// TIA Portal V19 export
FUNCTION_BLOCK "Positioning_EPOS_Machine_FB"   // FB55, LAD
TITLE = CLOSE LOOP POSITIONING AXIS WITH DRIVE S120 TEL.111 EPOS
// stored: Access Published, MemoryReserve 100, SetENOAutomatically false
   VAR_INPUT
      AreaInterface : "AreaInterface";
      ZSI : "udt_ZoneSafetyInterface";
      DSI : "udt_DeviceSafetyInterface";
      Drive : "TAx_DriveInterface";
      DataIn : "Positioning_EPOS_Machine_DataIn";
      CIn : "Positioning_EPOS_Machine_CIn";
      Config : "Positioning_EPOS_Machine_Config";
      HW_ID_TEL111 : HW_SUBMODULE;
   END_VAR
   VAR_OUTPUT
      MachineInterface { ExternalAccessible := 'False'; ExternalVisible := 'False'; ExternalWritable := 'False'} : "MachineInterface";
      DataOut : "Positioning_EPOS_Machine_DataOut";
      COut : "Positioning_EPOS_Machine_COut";
   END_VAR
   VAR_IN_OUT
      Par : "Positioning_EPOS_Machine_Par";
      Warning : "Positioning_EPOS_Machine_Wng";
      Alarm : "Positioning_EPOS_Machine_Alr";
   END_VAR
   VAR
      InitDone : Bool := FALSE;
      Status : Int;
      Diag : Struct
         S120 : "TO_Diagnostic";
      END_STRUCT;
      HMI : Struct
         Sts { S7_SetPoint := 'True'} : "UDT_HMI-Sts_PosEPOS-MchFB";
         B_Preset : Bool;
         PresetPosition : LReal;
         TargetPosition : LReal;
      END_STRUCT;
      Sts : Struct
         Standstill : Bool;
         AlarmPresence : Bool;
         WarningPresence : Bool;
         Gen_Cnd : Bool;
         Minus_Cnd : Bool;
         Plus_Cnd : Bool;
         Pos_Cnd : Bool;
         Preset_Cnd : Bool;
         InTargetPosition : Bool;
         Limits_SW_Active : Bool;
         Limits_EXT_Active : Bool;
         AxisModulo : LReal;
         ActualPosition : LReal;
         MissingToTarget : LReal;
         ActualVelocityRPM : LReal;
         ReductionRatio : LReal;
         ActualVelocity : LReal;
         S120 : Struct
            FaultActive : Bool;
            AlarmPresence : Bool;
            Standstill : Bool;
            IsRunningNegative : Bool;
            IsRunningPositive : Bool;
            MinusSWLim : Bool;
            PlusSWLim : Bool;
            MinusHWLim : Bool;
            PlusHWLim : Bool;
            TargetApply : Bool;
         END_STRUCT;
      END_STRUCT;
      Ctrl : Struct
         StopDueDoorOpeningRequest : Bool;
         StopAborting : Bool;
         SafeMotionEnable : Bool;
         StopInPhase : Bool;
         StopProgrammed : Bool;
         Preset : Bool;
         Minus_Man : Bool;
         Plus_Man : Bool;
         MoveToPos_Man : Bool;
         Minus_Aut : Bool;
         Plus_Aut : Bool;
         MoveToPos_Aut : Bool;
         MoveToPos : Bool;
         Minus_Vel : Bool;
         Plus_Vel : Bool;
         Fan : Bool;
         Pos : LReal;
         Vel : LReal;
         Acc : LReal;
         Dec : LReal;
         S120 : Struct
            Preset : Bool;
            Jog_Plus : Bool;
            Jog_Minus : Bool;
            Positioining : Bool;
            TargetPos : DInt;   // [LU] = Eng.Unit / 1000
         END_STRUCT;
      END_STRUCT;
      S120_SinaPos { S7_SetPoint := 'True'} : SinaPos;
      Fan_M : "Motor";
      WriteRefPos { S7_SetPoint := 'True'} : "RW_SINAMICS_Par";
      TON_DelayOFF { S7_SetPoint := 'True'} : TON_TIME;
      TON_ModeTimeOut { S7_SetPoint := 'True'} : TON_TIME;
      TON_NoPendingCmd : TON_TIME;
      TON_MinusCnd { S7_SetPoint := 'True'} : TON_TIME;
      TON_PlusCnd { S7_SetPoint := 'True'} : TON_TIME;
      TON_Fan_DelayOff : TON_TIME;
      TON_Brake_TimeOut : TON_TIME;
      TON_InTargetPosition { S7_SetPoint := 'True'} : TON_TIME;
      AUX : Struct
         PB_Minus : Bool;
         PB_Plus : Bool;
         PB_MoveToPos { ExternalAccessible := 'False'; ExternalVisible := 'False'; ExternalWritable := 'False'} : Bool;
         B_Preset { ExternalAccessible := 'False'; ExternalVisible := 'False'; ExternalWritable := 'False'} : Bool;
      END_STRUCT;
   END_VAR
   VAR_TEMP
      PE : Struct
         PB_Minus : Bool;
         PB_Plus : Bool;
         PB_MoveToPos : Bool;
         B_Preset : Bool;
      END_STRUCT;
      RETVAL : Int;
      Req : Bool;
      RemainingDistanceABS : LReal;
      LimitExceeds : Bool;
      UsePositionLimits : Bool;
      DriveSwitchOnInhibit : Bool;
   END_VAR
   VAR CONSTANT
      MODE_1_RELATIVE_POSITIONING : Int := 1;
      MODE_2_ABSOLUTE_POSITIONING : Int := 2;
      MODE_3_POS_AS_SETUP : Int := 3;
      MODE_4_HOMING_PROCEDURE : Int := 4;
      MODE_5_SET_HOME_POSITION : Int := 5;
      MODE_6_TRAVERSING_BLOCK : Int := 6;
      MODE_7_JOG : Int := 7;
      MODE_8_JOG_INCREMENTAL : Int := 8;
      STS_0_IDLE : Int := 0;
      STS_DIRECT_HOME : Int := 10;
      STS_MOVE_VEL : Int := 20;
      STS_POSITIONING_START : Int := 30;
      STS_STOP : Int := 90;
   END_VAR
   VAR_TEMP   // added for the SCL form of the ladder/FBD networks
      _w1 : Bool;
      _w2 : Bool;
      _w3 : Bool;
      _w4 : Bool;
   END_VAR
BEGIN

REGION Network 1 (SCL): Init

   IF NOT #InitDone THEN

       #InitDone := TRUE;

   END_IF;
END_REGION

REGION Network 2 (SCL): Reset
   IF #AreaInterface.RstAlarms THEN


       #Alarm.Ax_NotHomed := FALSE;
       #Alarm.HwLimitMinus := FALSE;
       #Alarm.HwLimitPlus := FALSE;


       #Warning.NotAutReady := FALSE;
       #Warning.Minus_CndMissing := FALSE;
       #Warning.Plus_CndMissing := FALSE;



   END_IF;
END_REGION

REGION Network 3: Reduction ratio calculation - Motor revolution -> position Eng Unit
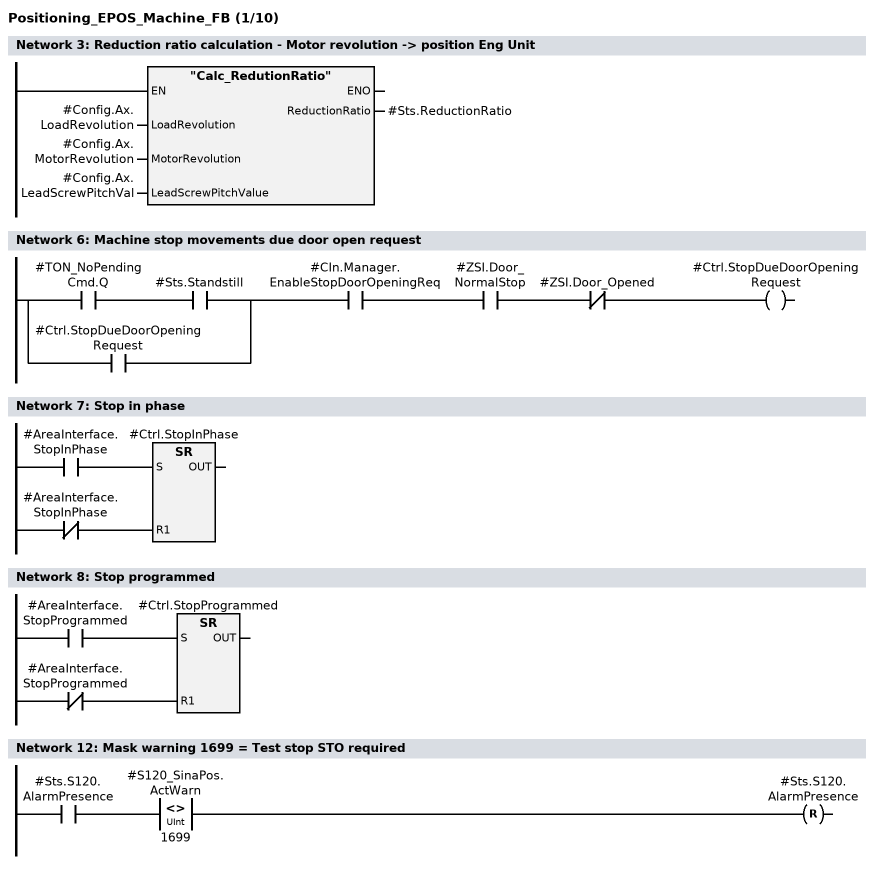
   RUNG wire#powerrail
      "Calc_RedutionRatio"(LoadRevolution := #Config.Ax.LoadRevolution, MotorRevolution := #Config.Ax.MotorRevolution, LeadScrewPitchValue := #Config.Ax.LeadScrewPitchVal, ReductionRatio => #Sts.ReductionRatio)
   END_RUNG
   // the same network as SCL:
   "Calc_RedutionRatio"(LoadRevolution := #Config.Ax.LoadRevolution,
                        MotorRevolution := #Config.Ax.MotorRevolution,
                        LeadScrewPitchValue := #Config.Ax.LeadScrewPitchVal,
                        ReductionRatio => #Sts.ReductionRatio);
END_REGION

REGION Network 4: >
END_REGION

REGION Network 5: <<< MACHINE STOP >>>
END_REGION

REGION Network 6: Machine stop movements due door open request
   RUNG wire#powerrail
      Contact( #TON_NoPendingCmd.Q )
      Contact( #Sts.Standstill )
      wire#w1
      Contact( #CIn.Manager.EnableStopDoorOpeningReq )
      Contact( #ZSI.Door_NormalStop )
      I_Contact( #ZSI.Door_Opened )
      Coil( #Ctrl.StopDueDoorOpeningRequest )
   END_RUNG
   RUNG wire#powerrail
      Contact( #Ctrl.StopDueDoorOpeningRequest )
   END_RUNG wire#w1
   // the same network as SCL:
   #Ctrl.StopDueDoorOpeningRequest := ((#TON_NoPendingCmd.Q AND #Sts.Standstill) OR #Ctrl.StopDueDoorOpeningRequest) AND #CIn.Manager.EnableStopDoorOpeningReq AND #ZSI.Door_NormalStop AND NOT #ZSI.Door_Opened;
END_REGION

REGION Network 7: Stop in phase
   RUNG wire#powerrail
      Contact( #AreaInterface.StopInPhase )
      S_SR(operand := #Ctrl.StopInPhase, r1 := wire#w1)
   END_RUNG
   RUNG wire#powerrail
      I_Contact( #AreaInterface.StopInPhase )
   END_RUNG wire#w1
   // the same network as SCL:
   IF #AreaInterface.StopInPhase THEN
       #Ctrl.StopInPhase := TRUE;   // SR flip-flop
   END_IF;
   IF NOT #AreaInterface.StopInPhase THEN #Ctrl.StopInPhase := FALSE; END_IF;
END_REGION

REGION Network 8: Stop programmed
   RUNG wire#powerrail
      Contact( #AreaInterface.StopProgrammed )
      S_SR(operand := #Ctrl.StopProgrammed, r1 := wire#w1)
   END_RUNG
   RUNG wire#powerrail
      I_Contact( #AreaInterface.StopProgrammed )
   END_RUNG wire#w1
   // the same network as SCL:
   IF #AreaInterface.StopProgrammed THEN
       #Ctrl.StopProgrammed := TRUE;   // SR flip-flop
   END_IF;
   IF NOT #AreaInterface.StopProgrammed THEN #Ctrl.StopProgrammed := FALSE; END_IF;
END_REGION

REGION Network 9: >
END_REGION

REGION Network 10 (SCL): Several status from FB
   // Axis modulo in Eng.Unit of position
   // 
   #Sts.AxisModulo := #Config.Ax.Modulo_S120_P2566 / 1000.0;


   // Position in Eng.Unit = Position in LU X 1000.
   //
   #Sts.ActualPosition := DINT_TO_LREAL(#S120_SinaPos.ActPosition) / 1000.0;

   // S120_SinaPos.ActVelocity = Current velocity (standardized 40000000h = 1073741824.0 dec = 100% = p2000)
   // Velocity in RPM
   // 
   #Sts.ActualVelocityRPM := DINT_TO_LREAL(#S120_SinaPos.ActVelocity) / 1073741824.0 * #Config.Ax.MaxRPM_S120_P2000;

   // Velocity in Eng.Unit / min
   #Sts.ActualVelocity := #Sts.ActualVelocityRPM * #Sts.ReductionRatio;


   #Sts.S120.IsRunningPositive := #S120_SinaPos.EPosZSW2.%X4;
   #Sts.S120.IsRunningNegative := #S120_SinaPos.EPosZSW2.%X5;

   #Sts.S120.MinusSWLim := #S120_SinaPos.EPosZSW2.%X6;
   #Sts.S120.PlusSWLim := #S120_SinaPos.EPosZSW2.%X7;

   #Sts.S120.MinusHWLim := #S120_SinaPos.EPosZSW1.%X8;
   #Sts.S120.PlusHWLim :=  #S120_SinaPos.EPosZSW1.%X9;


   #Sts.S120.FaultActive := #S120_SinaPos.ZSW1.%X3;
   #Sts.S120.AlarmPresence := #S120_SinaPos.ZSW1.%X7;
   #Sts.S120.Standstill := NOT #S120_SinaPos.EPosZSW1.%X4 AND NOT #S120_SinaPos.EPosZSW1.%X5 AND NOT #S120_SinaPos.EPosZSW2.%X4 AND NOT #S120_SinaPos.EPosZSW2.%X5;
END_REGION

REGION Network 11 (SCL): Drive Diagnostic
   #Diag.S120.DeviceType := 6;


   #Diag.S120.Drive_Message := 0;
   #Diag.S120.MessageType := 0;


   IF #Sts.S120.FaultActive THEN
       #Diag.S120.Drive_Message := #S120_SinaPos.ActFault;
       #Diag.S120.MessageType := 2;

   ELSIF #Sts.S120.AlarmPresence THEN
       #Diag.S120.Drive_Message := #S120_SinaPos.ActWarn;
       #Diag.S120.MessageType := 1;
   END_IF;
END_REGION

REGION Network 12: Mask warning 1699 = Test stop STO required
   RUNG wire#powerrail
      Contact( #Sts.S120.AlarmPresence )
      { S7_Templates := "SrcType := UInt" } NE_Contact(in1 := #S120_SinaPos.ActWarn, in2 := 1699)
      R_Coil( #Sts.S120.AlarmPresence )
   END_RUNG
   // the same network as SCL:
   IF #Sts.S120.AlarmPresence AND (#S120_SinaPos.ActWarn <> 1699) THEN
       #Sts.S120.AlarmPresence := FALSE;
   END_IF;
END_REGION

REGION Network 13: Drive / Axis Warnings
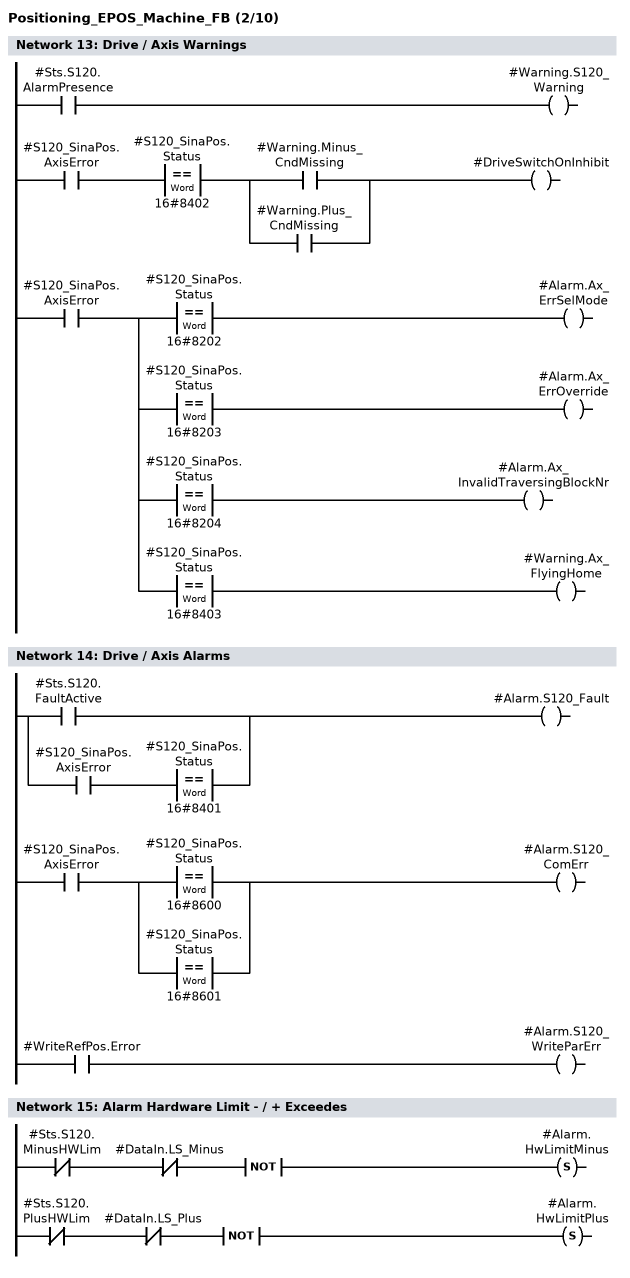
   RUNG wire#powerrail
      Contact( #Sts.S120.AlarmPresence )
      Coil( #Warning.S120_Warning )
   END_RUNG
   RUNG wire#powerrail
      Contact( #S120_SinaPos.AxisError )
      { S7_Templates := "SrcType := Word" } EQ_Contact(in1 := #S120_SinaPos.Status, in2 := 16#8402)
      wire#w1
      Contact( #Warning.Minus_CndMissing )
      wire#w2
      Coil( #DriveSwitchOnInhibit )
   END_RUNG
   RUNG wire#w1
      Contact( #Warning.Plus_CndMissing )
   END_RUNG wire#w2
   RUNG wire#powerrail
      Contact( #S120_SinaPos.AxisError )
      wire#w3
      { S7_Templates := "SrcType := Word" } EQ_Contact(in1 := #S120_SinaPos.Status, in2 := 16#8202)
      Coil( #Alarm.Ax_ErrSelMode )
   END_RUNG
   RUNG wire#w3
      { S7_Templates := "SrcType := Word" } EQ_Contact(in1 := #S120_SinaPos.Status, in2 := 16#8203)
      Coil( #Alarm.Ax_ErrOverride )
   END_RUNG
   RUNG wire#w3
      { S7_Templates := "SrcType := Word" } EQ_Contact(in1 := #S120_SinaPos.Status, in2 := 16#8204)
      Coil( #Alarm.Ax_InvalidTraversingBlockNr )
   END_RUNG
   RUNG wire#w3
      { S7_Templates := "SrcType := Word" } EQ_Contact(in1 := #S120_SinaPos.Status, in2 := 16#8403)
      Coil( #Warning.Ax_FlyingHome )
   END_RUNG
   // the same network as SCL:
   #Warning.S120_Warning := #Sts.S120.AlarmPresence;
   #DriveSwitchOnInhibit := #S120_SinaPos.AxisError AND (#S120_SinaPos.Status = 16#8402) AND (#Warning.Minus_CndMissing OR #Warning.Plus_CndMissing);
   #Alarm.Ax_ErrSelMode := #S120_SinaPos.AxisError AND (#S120_SinaPos.Status = 16#8202);
   #Alarm.Ax_ErrOverride := #S120_SinaPos.AxisError AND (#S120_SinaPos.Status = 16#8203);
   #Alarm.Ax_InvalidTraversingBlockNr := #S120_SinaPos.AxisError AND (#S120_SinaPos.Status = 16#8204);
   #Warning.Ax_FlyingHome := #S120_SinaPos.AxisError AND (#S120_SinaPos.Status = 16#8403);
END_REGION

REGION Network 14: Drive / Axis Alarms
   RUNG wire#powerrail
      Contact( #Sts.S120.FaultActive )
      wire#w1
      Coil( #Alarm.S120_Fault )
   END_RUNG
   RUNG wire#powerrail
      Contact( #S120_SinaPos.AxisError )
      { S7_Templates := "SrcType := Word" } EQ_Contact(in1 := #S120_SinaPos.Status, in2 := 16#8401)
   END_RUNG wire#w1
   RUNG wire#powerrail
      Contact( #S120_SinaPos.AxisError )
      wire#w2
      { S7_Templates := "SrcType := Word" } EQ_Contact(in1 := #S120_SinaPos.Status, in2 := 16#8600)
      wire#w3
      Coil( #Alarm.S120_ComErr )
   END_RUNG
   RUNG wire#w2
      { S7_Templates := "SrcType := Word" } EQ_Contact(in1 := #S120_SinaPos.Status, in2 := 16#8601)
   END_RUNG wire#w3
   RUNG wire#powerrail
      Contact( #WriteRefPos.Error )
      Coil( #Alarm.S120_WriteParErr )
   END_RUNG
   // the same network as SCL:
   #Alarm.S120_Fault := #Sts.S120.FaultActive OR (#S120_SinaPos.AxisError AND (#S120_SinaPos.Status = 16#8401));
   #Alarm.S120_ComErr := #S120_SinaPos.AxisError AND ((#S120_SinaPos.Status = 16#8600) OR (#S120_SinaPos.Status = 16#8601));
   #Alarm.S120_WriteParErr := #WriteRefPos.Error;
END_REGION

REGION Network 15: Alarm Hardware Limit - / + Exceedes
   RUNG wire#powerrail
      I_Contact( #Sts.S120.MinusHWLim )
      I_Contact( #DataIn.LS_Minus )
      Not()
      S_Coil( #Alarm.HwLimitMinus )
   END_RUNG
   RUNG wire#powerrail
      I_Contact( #Sts.S120.PlusHWLim )
      I_Contact( #DataIn.LS_Plus )
      Not()
      S_Coil( #Alarm.HwLimitPlus )
   END_RUNG
   // the same network as SCL:
   IF NOT (NOT #Sts.S120.MinusHWLim AND NOT #DataIn.LS_Minus) THEN #Alarm.HwLimitMinus := TRUE; END_IF;
   IF NOT (NOT #Sts.S120.PlusHWLim AND NOT #DataIn.LS_Plus) THEN #Alarm.HwLimitPlus := TRUE; END_IF;
END_REGION

REGION Network 16: Warning software limit - / + Exceedes
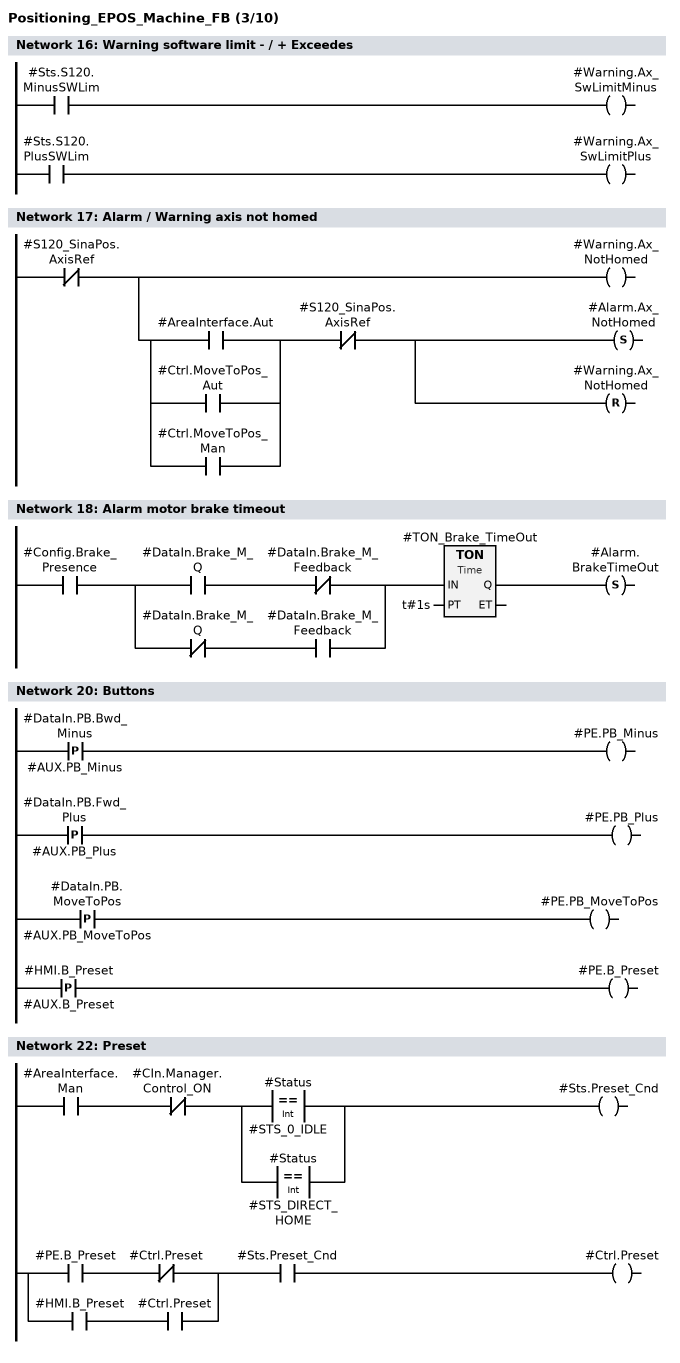
   RUNG wire#powerrail
      Contact( #Sts.S120.MinusSWLim )
      Coil( #Warning.Ax_SwLimitMinus )
   END_RUNG
   RUNG wire#powerrail
      Contact( #Sts.S120.PlusSWLim )
      Coil( #Warning.Ax_SwLimitPlus )
   END_RUNG
   // the same network as SCL:
   #Warning.Ax_SwLimitMinus := #Sts.S120.MinusSWLim;
   #Warning.Ax_SwLimitPlus := #Sts.S120.PlusSWLim;
END_REGION

REGION Network 17: Alarm / Warning axis not homed
   RUNG wire#powerrail
      I_Contact( #S120_SinaPos.AxisRef )
      wire#w1
      Coil( #Warning.Ax_NotHomed )
   END_RUNG
   RUNG wire#w1
      Contact( #AreaInterface.Aut )
      wire#w2
      I_Contact( #S120_SinaPos.AxisRef )
      wire#w3
      S_Coil( #Alarm.Ax_NotHomed )
   END_RUNG
   RUNG wire#w1
      Contact( #Ctrl.MoveToPos_Aut )
   END_RUNG wire#w2
   RUNG wire#w1
      Contact( #Ctrl.MoveToPos_Man )
   END_RUNG wire#w2
   RUNG wire#w3
      R_Coil( #Warning.Ax_NotHomed )
   END_RUNG
   // the same network as SCL:
   #Warning.Ax_NotHomed := NOT #S120_SinaPos.AxisRef;
   IF NOT #S120_SinaPos.AxisRef AND (#AreaInterface.Aut OR #Ctrl.MoveToPos_Aut OR #Ctrl.MoveToPos_Man) AND NOT #S120_SinaPos.AxisRef THEN
       #Alarm.Ax_NotHomed := TRUE;
       #Warning.Ax_NotHomed := FALSE;
   END_IF;
END_REGION

REGION Network 18: Alarm motor brake timeout
   RUNG wire#powerrail
      Contact( #Config.Brake_Presence )
      wire#w1
      Contact( #DataIn.Brake_M_Q )
      I_Contact( #DataIn.Brake_M_Feedback )
      wire#w2
      { S7_Templates := "time_type := Time" } #TON_Brake_TimeOut.TON(pt := t#1s, et =>)
      S_Coil( #Alarm.BrakeTimeOut )
   END_RUNG
   RUNG wire#w1
      I_Contact( #DataIn.Brake_M_Q )
      Contact( #DataIn.Brake_M_Feedback )
   END_RUNG wire#w2
   // the same network as SCL:
   #TON_Brake_TimeOut(IN := #Config.Brake_Presence AND ((#DataIn.Brake_M_Q AND NOT #DataIn.Brake_M_Feedback) OR (NOT #DataIn.Brake_M_Q AND #DataIn.Brake_M_Feedback)),   // TON
                      PT := t#1s);
   IF #TON_Brake_TimeOut.Q THEN #Alarm.BrakeTimeOut := TRUE; END_IF;
END_REGION

REGION Network 19: >
END_REGION

REGION Network 20: Buttons
   RUNG wire#powerrail
      P_Contact(operand := #DataIn.PB.Bwd_Minus, bit := #AUX.PB_Minus)
      Coil( #PE.PB_Minus )
   END_RUNG
   RUNG wire#powerrail
      P_Contact(operand := #DataIn.PB.Fwd_Plus, bit := #AUX.PB_Plus)
      Coil( #PE.PB_Plus )
   END_RUNG
   RUNG wire#powerrail
      P_Contact(operand := #DataIn.PB.MoveToPos, bit := #AUX.PB_MoveToPos)
      Coil( #PE.PB_MoveToPos )
   END_RUNG
   RUNG wire#powerrail
      P_Contact(operand := #HMI.B_Preset, bit := #AUX.B_Preset)
      Coil( #PE.B_Preset )
   END_RUNG
   // the same network as SCL:
   #_w1 := #DataIn.PB.Bwd_Minus AND NOT #AUX.PB_Minus;   // rising edge of #DataIn.PB.Bwd_Minus
   #AUX.PB_Minus := #DataIn.PB.Bwd_Minus;
   #PE.PB_Minus := #_w1;
   #_w2 := #DataIn.PB.Fwd_Plus AND NOT #AUX.PB_Plus;   // rising edge of #DataIn.PB.Fwd_Plus
   #AUX.PB_Plus := #DataIn.PB.Fwd_Plus;
   #PE.PB_Plus := #_w2;
   #_w3 := #DataIn.PB.MoveToPos AND NOT #AUX.PB_MoveToPos;   // rising edge of #DataIn.PB.MoveToPos
   #AUX.PB_MoveToPos := #DataIn.PB.MoveToPos;
   #PE.PB_MoveToPos := #_w3;
   #_w4 := #HMI.B_Preset AND NOT #AUX.B_Preset;   // rising edge of #HMI.B_Preset
   #AUX.B_Preset := #HMI.B_Preset;
   #PE.B_Preset := #_w4;
END_REGION

REGION Network 21: >
END_REGION

REGION Network 22: Preset
   RUNG wire#powerrail
      Contact( #AreaInterface.Man )
      I_Contact( #CIn.Manager.Control_ON )
      wire#w1
      { S7_Templates := "SrcType := Int" } EQ_Contact(in1 := #Status, in2 := #STS_0_IDLE)
      wire#w2
      Coil( #Sts.Preset_Cnd )
   END_RUNG
   RUNG wire#w1
      { S7_Templates := "SrcType := Int" } EQ_Contact(in1 := #Status, in2 := #STS_DIRECT_HOME)
   END_RUNG wire#w2
   RUNG wire#powerrail
      Contact( #PE.B_Preset )
      I_Contact( #Ctrl.Preset )
      wire#w3
      Contact( #Sts.Preset_Cnd )
      Coil( #Ctrl.Preset )
   END_RUNG
   RUNG wire#powerrail
      Contact( #HMI.B_Preset )
      Contact( #Ctrl.Preset )
   END_RUNG wire#w3
   // the same network as SCL:
   #Sts.Preset_Cnd := #AreaInterface.Man AND NOT #CIn.Manager.Control_ON AND ((#Status = #STS_0_IDLE) OR (#Status = #STS_DIRECT_HOME));
   #Ctrl.Preset := ((#PE.B_Preset AND NOT #Ctrl.Preset) OR (#HMI.B_Preset AND #Ctrl.Preset)) AND #Sts.Preset_Cnd;
END_REGION

REGION Network 23: Man
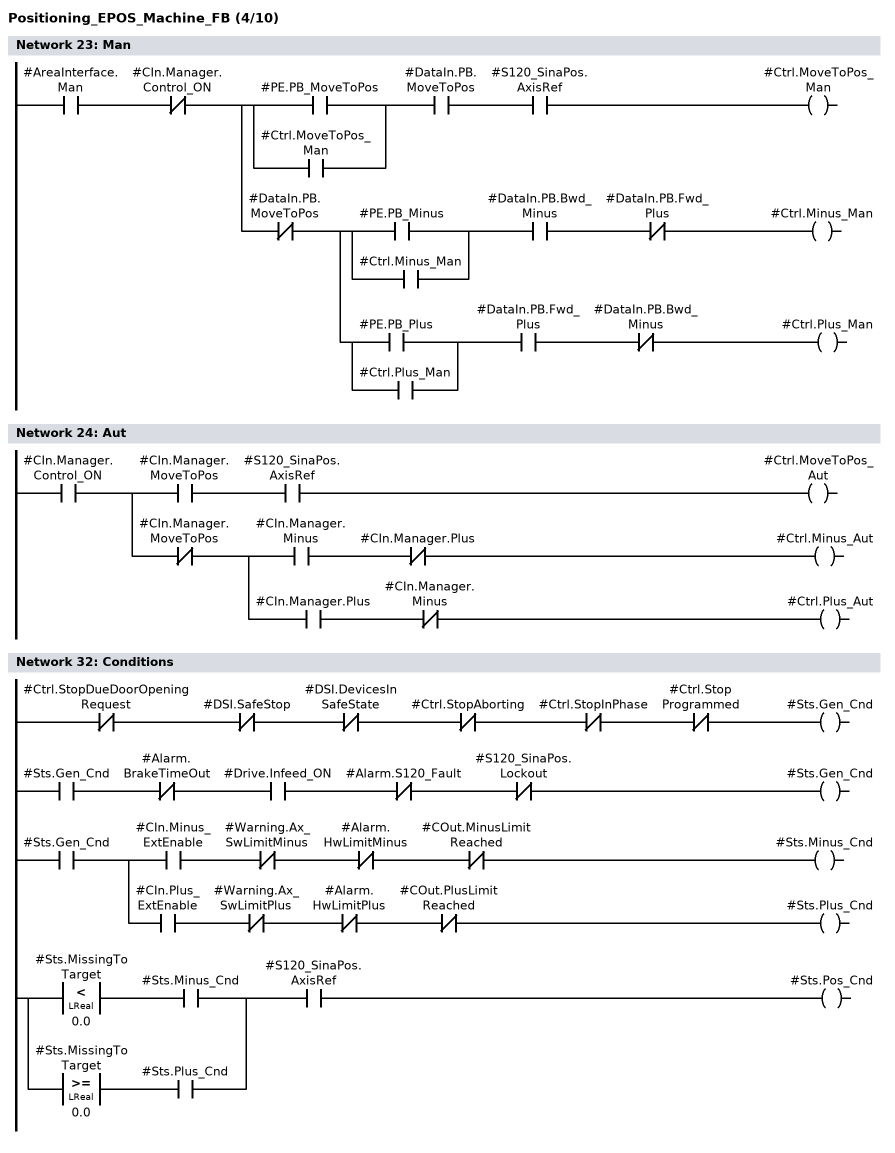
   RUNG wire#powerrail
      Contact( #AreaInterface.Man )
      I_Contact( #CIn.Manager.Control_ON )
      wire#w1
      Contact( #PE.PB_MoveToPos )
      wire#w2
      Contact( #DataIn.PB.MoveToPos )
      Contact( #S120_SinaPos.AxisRef )
      Coil( #Ctrl.MoveToPos_Man )
   END_RUNG
   RUNG wire#w1
      Contact( #Ctrl.MoveToPos_Man )
   END_RUNG wire#w2
   RUNG wire#w1
      I_Contact( #DataIn.PB.MoveToPos )
      wire#w3
      Contact( #PE.PB_Minus )
      wire#w4
      Contact( #DataIn.PB.Bwd_Minus )
      I_Contact( #DataIn.PB.Fwd_Plus )
      Coil( #Ctrl.Minus_Man )
   END_RUNG
   RUNG wire#w3
      Contact( #Ctrl.Minus_Man )
   END_RUNG wire#w4
   RUNG wire#w3
      Contact( #PE.PB_Plus )
      wire#w5
      Contact( #DataIn.PB.Fwd_Plus )
      I_Contact( #DataIn.PB.Bwd_Minus )
      Coil( #Ctrl.Plus_Man )
   END_RUNG
   RUNG wire#w3
      Contact( #Ctrl.Plus_Man )
   END_RUNG wire#w5
   // the same network as SCL:
   #_w1 := #AreaInterface.Man AND NOT #CIn.Manager.Control_ON;
   #Ctrl.MoveToPos_Man := #_w1 AND (#PE.PB_MoveToPos OR #Ctrl.MoveToPos_Man) AND #DataIn.PB.MoveToPos AND #S120_SinaPos.AxisRef;
   #_w2 := #_w1 AND NOT #DataIn.PB.MoveToPos;
   #Ctrl.Minus_Man := #_w2 AND (#PE.PB_Minus OR #Ctrl.Minus_Man) AND #DataIn.PB.Bwd_Minus AND NOT #DataIn.PB.Fwd_Plus;
   #Ctrl.Plus_Man := #_w2 AND (#PE.PB_Plus OR #Ctrl.Plus_Man) AND #DataIn.PB.Fwd_Plus AND NOT #DataIn.PB.Bwd_Minus;
END_REGION

REGION Network 24: Aut
   RUNG wire#powerrail
      Contact( #CIn.Manager.Control_ON )
      wire#w1
      Contact( #CIn.Manager.MoveToPos )
      Contact( #S120_SinaPos.AxisRef )
      Coil( #Ctrl.MoveToPos_Aut )
   END_RUNG
   RUNG wire#w1
      I_Contact( #CIn.Manager.MoveToPos )
      wire#w2
      Contact( #CIn.Manager.Minus )
      I_Contact( #CIn.Manager.Plus )
      Coil( #Ctrl.Minus_Aut )
   END_RUNG
   RUNG wire#w2
      Contact( #CIn.Manager.Plus )
      I_Contact( #CIn.Manager.Minus )
      Coil( #Ctrl.Plus_Aut )
   END_RUNG
   // the same network as SCL:
   #Ctrl.MoveToPos_Aut := #CIn.Manager.Control_ON AND #CIn.Manager.MoveToPos AND #S120_SinaPos.AxisRef;
   #_w1 := #CIn.Manager.Control_ON AND NOT #CIn.Manager.MoveToPos;
   #Ctrl.Minus_Aut := #_w1 AND #CIn.Manager.Minus AND NOT #CIn.Manager.Plus;
   #Ctrl.Plus_Aut := #_w1 AND #CIn.Manager.Plus AND NOT #CIn.Manager.Minus;
END_REGION

REGION Network 25: >
END_REGION

REGION Network 26 (SCL): Position Limits
   #COut.MinPosition := -999999999.99;
   #COut.MaxPosition := +999999999.99;

   #COut.MinusLsSwReached := FALSE;
   #COut.PlusLsSwReached := FALSE;
   #COut.MinusLimitReached := FALSE;
   #COut.PlusLimitReached := FALSE;

   #Sts.Limits_SW_Active := FALSE;
   #Sts.Limits_EXT_Active := FALSE;


   IF #S120_SinaPos.AxisRef
   THEN

       #Sts.Limits_SW_Active := #Config.Ax.SwLimMinus_S120_P2580 < #Config.Ax.SwLimPlus_S120_P2581;

       //.. If software limits are enabled...
       //
       IF #Sts.Limits_SW_Active
       THEN


           // Software limit Minus reached or exceeds
           // 
           #RemainingDistanceABS := ABS("M_PosAMinusPosB"(PosA := #Sts.ActualPosition, PosB := #Config.Ax.SwLimMinus_S120_P2580, MODULE := #Sts.AxisModulo));

           #LimitExceeds := "M_CmpLT"(Xa := #Sts.ActualPosition, Xb := #Config.Ax.SwLimMinus_S120_P2580, MODULE := #Sts.AxisModulo);

           #COut.MinusLsSwReached := (#RemainingDistanceABS <= #Par.PosTolerance) OR #LimitExceeds;


           // Software limit Plus reached or exceeds
           // 
           #RemainingDistanceABS := ABS("M_PosAMinusPosB"(PosA := #Sts.ActualPosition, PosB := #Config.Ax.SwLimPlus_S120_P2581, MODULE := #Sts.AxisModulo));

           #LimitExceeds := "M_CmpGT"(Xa := #Sts.ActualPosition, Xb :=#Config.Ax.SwLimPlus_S120_P2581, MODULE := #Sts.AxisModulo);

           #COut.PlusLsSwReached := (#RemainingDistanceABS <= #Par.PosTolerance) OR #LimitExceeds;


           // Set general Min / Max position limit
           // 
           #COut.MinPosition := "M_PosAPlusCostB"(PosA := #Config.Ax.SwLimMinus_S120_P2580, CostB := (#Par.PosTolerance / 2), MODULE := #Sts.AxisModulo);
           #COut.MaxPosition := "M_PosAMinusCostB"(PosA := #Config.Ax.SwLimPlus_S120_P2581, CostB := (#Par.PosTolerance / 2), MODULE := #Sts.AxisModulo);


       END_IF;

       //.. IF External MIN limit set..
       //
       IF #CIn.PositionLimits.EnableMin
       THEN
           #Sts.Limits_EXT_Active := TRUE;

           #RemainingDistanceABS := ABS("M_PosAMinusPosB"(PosA := #Sts.ActualPosition, PosB := #CIn.PositionLimits.PosMin, MODULE := #Sts.AxisModulo));

           #LimitExceeds := "M_CmpLT"(Xa := #Sts.ActualPosition, Xb := #CIn.PositionLimits.PosMin, MODULE := #Sts.AxisModulo);

           #COut.MinusLimitReached := (#RemainingDistanceABS <= #Par.PosTolerance) OR #LimitExceeds;

           // Update general MIN limit
           // 
           IF "M_CmpGT"(Xa := #CIn.PositionLimits.PosMin, Xb := #COut.MinPosition, MODULE := #Sts.AxisModulo)
           THEN
               #COut.MinPosition := #CIn.PositionLimits.PosMin;
           END_IF;
       END_IF;


       //.. IF External MAX limit set..
       //
       IF #CIn.PositionLimits.EnableMax
       THEN
           #Sts.Limits_EXT_Active := TRUE;

           #RemainingDistanceABS := ABS("M_PosAMinusPosB"(PosA := #Sts.ActualPosition, PosB := #CIn.PositionLimits.PosMax, MODULE := #Sts.AxisModulo));

           #LimitExceeds := "M_CmpGT"(Xa := #Sts.ActualPosition, Xb := #CIn.PositionLimits.PosMax, MODULE := #Sts.AxisModulo);

           #COut.PlusLimitReached := (#RemainingDistanceABS <= #Par.PosTolerance) OR #LimitExceeds;


           // Update general MAX limit
           // 
           IF "M_CmpLT"(Xa := #CIn.PositionLimits.PosMax, Xb := #COut.MaxPosition, MODULE := #Sts.AxisModulo)
           THEN
               #COut.MaxPosition := #CIn.PositionLimits.PosMax;
           END_IF;

       END_IF;

   END_IF;


   #UsePositionLimits := #Sts.Limits_SW_Active OR #Sts.Limits_EXT_Active;
END_REGION

REGION Network 27 (SCL): Target Position
   // Target position choose
   //


   IF #CIn.Manager.Control_ON
   THEN

       #Ctrl.Pos := #CIn.Manager.Pos;


       IF #Ctrl.Minus_Aut AND #UsePositionLimits
       THEN
           #Ctrl.Pos := #COut.MinPosition;


       ELSIF #Ctrl.Plus_Aut AND #UsePositionLimits
       THEN
           #Ctrl.Pos := #COut.MaxPosition;
       END_IF;


       #HMI.TargetPosition := #Ctrl.Pos;



   ELSIF #Ctrl.MoveToPos_Man
   THEN

       #Ctrl.Pos := #HMI.TargetPosition;


   ELSIF #Ctrl.Minus_Man AND #UsePositionLimits
   THEN
       #Ctrl.Pos := #COut.MinPosition;
       #HMI.TargetPosition := #Ctrl.Pos;

   ELSIF #Ctrl.Plus_Man AND #UsePositionLimits
   THEN

       #Ctrl.Pos := #COut.MaxPosition;
       #HMI.TargetPosition := #Ctrl.Pos;

   END_IF;



   // Check Target position within limits
   // 

   IF #UsePositionLimits THEN


       // Target position exceeds MIN limit
       // 
       #LimitExceeds := "M_CmpLT"(Xa := #Ctrl.Pos, Xb := #COut.MinPosition, MODULE := #Sts.AxisModulo);
       IF #LimitExceeds THEN
           #Ctrl.Pos := #COut.MinPosition;
       END_IF;


       // Target position exceeds MAX limit
       //  
       #LimitExceeds := "M_CmpGT"(Xa := #Ctrl.Pos, Xb := #COut.MaxPosition, MODULE := #Sts.AxisModulo);
       IF #LimitExceeds THEN
           #Ctrl.Pos := #COut.MaxPosition;
       END_IF;

   END_IF;
END_REGION

REGION Network 28 (SCL): Check missing position to reach the target
   #Sts.MissingToTarget := "M_PosAMinusPosB"(PosA := #Ctrl.Pos, PosB := #Sts.ActualPosition, MODULE := #Sts.AxisModulo);
END_REGION

REGION Network 29 (SCL): Status axis in target position

   #TON_InTargetPosition(IN := ABS(#Sts.MissingToTarget) <= #Par.PosTolerance, PT := #Par.DelayInPosition);

   #Sts.InTargetPosition := #TON_InTargetPosition.Q AND #S120_SinaPos.AxisRef AND (#S120_SinaPos.AxisPosOk OR NOT #Ctrl.S120.Positioining);
END_REGION

REGION Network 30 (SCL): Target Velocity / Acc / Dec
   #Ctrl.Vel := 0.0;

   IF #CIn.Manager.Control_ON THEN

       #Ctrl.Vel := #CIn.Manager.Vel;
       #Ctrl.Acc := #CIn.Manager.Acc;
       #Ctrl.Dec := #CIn.Manager.Dec;


   ELSIF #Ctrl.Minus_Man OR #Ctrl.Plus_Man OR #Ctrl.MoveToPos_Man THEN

       #Ctrl.Vel := #Par.Man_Vel;
       #Ctrl.Acc := #Par.Man_Acc;
       #Ctrl.Dec := #Par.Man_Dec;

   END_IF;


   //---   

   // Dynamics limiting
   // 
   #Ctrl.Vel := MIN(IN1 := #Ctrl.Vel, IN2 := #Config.Ax.MaxVel_S120_P2571);
   #Ctrl.Acc := MIN(IN1 := #Ctrl.Acc, IN2 := #Config.Ax.MaxAcc_S120_P2572);
   #Ctrl.Dec := MIN(IN1 := #Ctrl.Dec, IN2 := #Config.Ax.MaxDec_S120_P2573);

   //---

   // SLS velocity limit
   //  
   IF #ZSI.Door_Opened AND #Ctrl.Vel > #Config.SLS_Vel THEN
       #Ctrl.Vel := #Config.SLS_Vel;
   END_IF;

   // Brake not open... Velocity  = 0.0
   // 
   IF #Config.Brake_Presence AND NOT #DataIn.Brake_M_Feedback THEN
       #Ctrl.Vel := 0.0;
   END_IF;


   #COut.MaxVelocity := #Config.Ax.MaxVel_S120_P2571;
END_REGION

REGION Network 31: >
END_REGION

REGION Network 32: Conditions
   RUNG wire#powerrail
      I_Contact( #Ctrl.StopDueDoorOpeningRequest )
      I_Contact( #DSI.SafeStop )
      I_Contact( #DSI.DevicesInSafeState )
      I_Contact( #Ctrl.StopAborting )
      I_Contact( #Ctrl.StopInPhase )
      I_Contact( #Ctrl.StopProgrammed )
      Coil( #Sts.Gen_Cnd )
   END_RUNG
   RUNG wire#powerrail
      Contact( #Sts.Gen_Cnd )
      I_Contact( #Alarm.BrakeTimeOut )
      Contact( #Drive.Infeed_ON )
      I_Contact( #Alarm.S120_Fault )
      I_Contact( #S120_SinaPos.Lockout )
      Coil( #Sts.Gen_Cnd )
   END_RUNG
   RUNG wire#powerrail
      Contact( #Sts.Gen_Cnd )
      wire#w1
      Contact( #CIn.Minus_ExtEnable )
      I_Contact( #Warning.Ax_SwLimitMinus )
      I_Contact( #Alarm.HwLimitMinus )
      I_Contact( #COut.MinusLimitReached )
      Coil( #Sts.Minus_Cnd )
   END_RUNG
   RUNG wire#w1
      Contact( #CIn.Plus_ExtEnable )
      I_Contact( #Warning.Ax_SwLimitPlus )
      I_Contact( #Alarm.HwLimitPlus )
      I_Contact( #COut.PlusLimitReached )
      Coil( #Sts.Plus_Cnd )
   END_RUNG
   RUNG wire#powerrail
      { S7_Templates := "SrcType := LReal" } LT_Contact(in1 := #Sts.MissingToTarget, in2 := 0.0)
      Contact( #Sts.Minus_Cnd )
      wire#w2
      Contact( #S120_SinaPos.AxisRef )
      Coil( #Sts.Pos_Cnd )
   END_RUNG
   RUNG wire#powerrail
      { S7_Templates := "SrcType := LReal" } GE_Contact(in1 := #Sts.MissingToTarget, in2 := 0.0)
      Contact( #Sts.Plus_Cnd )
   END_RUNG wire#w2
   // the same network as SCL:
   #Sts.Gen_Cnd := NOT #Ctrl.StopDueDoorOpeningRequest AND NOT #DSI.SafeStop AND NOT #DSI.DevicesInSafeState AND NOT #Ctrl.StopAborting AND NOT #Ctrl.StopInPhase AND NOT #Ctrl.StopProgrammed;
   #Sts.Gen_Cnd := #Sts.Gen_Cnd AND NOT #Alarm.BrakeTimeOut AND #Drive.Infeed_ON AND NOT #Alarm.S120_Fault AND NOT #S120_SinaPos.Lockout;
   #Sts.Minus_Cnd := #Sts.Gen_Cnd AND #CIn.Minus_ExtEnable AND NOT #Warning.Ax_SwLimitMinus AND NOT #Alarm.HwLimitMinus AND NOT #COut.MinusLimitReached;
   #Sts.Plus_Cnd := #Sts.Gen_Cnd AND #CIn.Plus_ExtEnable AND NOT #Warning.Ax_SwLimitPlus AND NOT #Alarm.HwLimitPlus AND NOT #COut.PlusLimitReached;
   #Sts.Pos_Cnd := (((#Sts.MissingToTarget < 0.0) AND #Sts.Minus_Cnd) OR ((#Sts.MissingToTarget >= 0.0) AND #Sts.Plus_Cnd)) AND #S120_SinaPos.AxisRef;
END_REGION

REGION Network 33: >
END_REGION

REGION Network 34: <<< S120 EPOS >>>
END_REGION

REGION Network 35: S120 EPOS - Controls
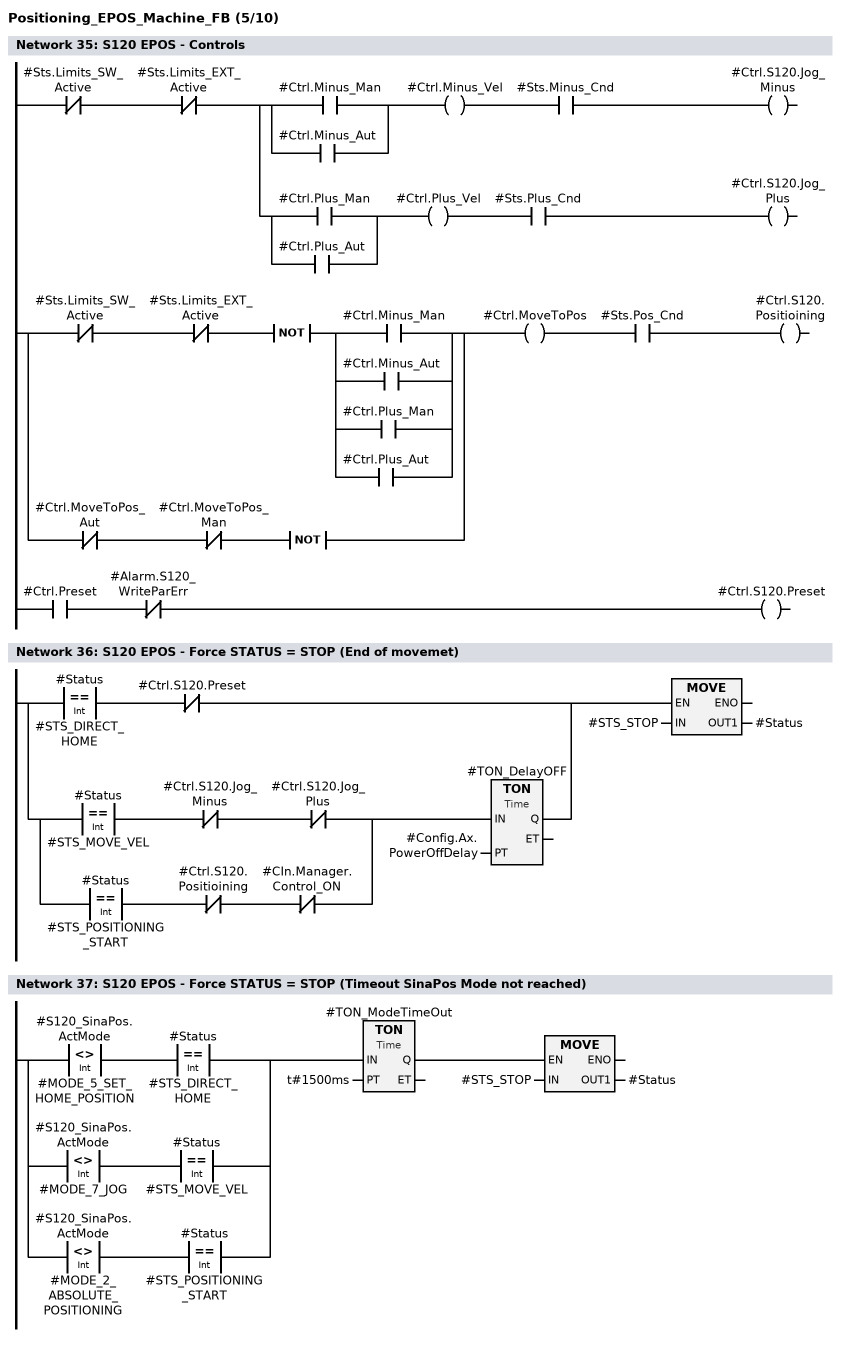
   RUNG wire#powerrail
      I_Contact( #Sts.Limits_SW_Active )
      I_Contact( #Sts.Limits_EXT_Active )
      wire#w1
      Contact( #Ctrl.Minus_Man )
      wire#w2
      Coil( #Ctrl.Minus_Vel )
      Contact( #Sts.Minus_Cnd )
      Coil( #Ctrl.S120.Jog_Minus )
   END_RUNG
   RUNG wire#w1
      Contact( #Ctrl.Minus_Aut )
   END_RUNG wire#w2
   RUNG wire#w1
      Contact( #Ctrl.Plus_Man )
      wire#w3
      Coil( #Ctrl.Plus_Vel )
      Contact( #Sts.Plus_Cnd )
      Coil( #Ctrl.S120.Jog_Plus )
   END_RUNG
   RUNG wire#w1
      Contact( #Ctrl.Plus_Aut )
   END_RUNG wire#w3
   RUNG wire#powerrail
      I_Contact( #Sts.Limits_SW_Active )
      I_Contact( #Sts.Limits_EXT_Active )
      Not()
      wire#w4
      Contact( #Ctrl.Minus_Man )
      wire#w5
      Coil( #Ctrl.MoveToPos )
      Contact( #Sts.Pos_Cnd )
      Coil( #Ctrl.S120.Positioining )
   END_RUNG
   RUNG wire#w4
      Contact( #Ctrl.Minus_Aut )
   END_RUNG wire#w5
   RUNG wire#w4
      Contact( #Ctrl.Plus_Man )
   END_RUNG wire#w5
   RUNG wire#w4
      Contact( #Ctrl.Plus_Aut )
   END_RUNG wire#w5
   RUNG wire#powerrail
      I_Contact( #Ctrl.MoveToPos_Aut )
      I_Contact( #Ctrl.MoveToPos_Man )
      Not()
   END_RUNG wire#w5
   RUNG wire#powerrail
      Contact( #Ctrl.Preset )
      I_Contact( #Alarm.S120_WriteParErr )
      Coil( #Ctrl.S120.Preset )
   END_RUNG
   // the same network as SCL:
   #_w1 := NOT #Sts.Limits_SW_Active AND NOT #Sts.Limits_EXT_Active;
   #Ctrl.Minus_Vel := #_w1 AND (#Ctrl.Minus_Man OR #Ctrl.Minus_Aut);
   #Ctrl.S120.Jog_Minus := #Ctrl.Minus_Vel AND #Sts.Minus_Cnd;
   #Ctrl.Plus_Vel := #_w1 AND (#Ctrl.Plus_Man OR #Ctrl.Plus_Aut);
   #Ctrl.S120.Jog_Plus := #Ctrl.Plus_Vel AND #Sts.Plus_Cnd;
   #Ctrl.MoveToPos := (NOT (NOT #Sts.Limits_SW_Active AND NOT #Sts.Limits_EXT_Active) AND (#Ctrl.Minus_Man OR #Ctrl.Minus_Aut OR #Ctrl.Plus_Man OR #Ctrl.Plus_Aut)) OR NOT (NOT #Ctrl.MoveToPos_Aut AND NOT #Ctrl.MoveToPos_Man);
   #Ctrl.S120.Positioining := #Ctrl.MoveToPos AND #Sts.Pos_Cnd;
   #Ctrl.S120.Preset := #Ctrl.Preset AND NOT #Alarm.S120_WriteParErr;
END_REGION

REGION Network 36: S120 EPOS - Force STATUS = STOP (End of movemet)
   RUNG wire#powerrail
      { S7_Templates := "SrcType := Int" } EQ_Contact(in1 := #Status, in2 := #STS_DIRECT_HOME)
      I_Contact( #Ctrl.S120.Preset )
      wire#w1
      Move(in := #STS_STOP, out1 => #Status)
   END_RUNG
   RUNG wire#powerrail
      { S7_Templates := "SrcType := Int" } EQ_Contact(in1 := #Status, in2 := #STS_MOVE_VEL)
      I_Contact( #Ctrl.S120.Jog_Minus )
      I_Contact( #Ctrl.S120.Jog_Plus )
      wire#w2
      { S7_Templates := "time_type := Time" } #TON_DelayOFF.TON(pt := #Config.Ax.PowerOffDelay, et =>)
   END_RUNG wire#w1
   RUNG wire#powerrail
      { S7_Templates := "SrcType := Int" } EQ_Contact(in1 := #Status, in2 := #STS_POSITIONING_START)
      I_Contact( #Ctrl.S120.Positioining )
      I_Contact( #CIn.Manager.Control_ON )
   END_RUNG wire#w2
   // the same network as SCL:
   #TON_DelayOFF(IN := ((#Status = #STS_MOVE_VEL) AND NOT #Ctrl.S120.Jog_Minus AND NOT #Ctrl.S120.Jog_Plus) OR ((#Status = #STS_POSITIONING_START) AND NOT #Ctrl.S120.Positioining AND NOT #CIn.Manager.Control_ON),   // TON
                 PT := #Config.Ax.PowerOffDelay);
   IF ((#Status = #STS_DIRECT_HOME) AND NOT #Ctrl.S120.Preset) OR #TON_DelayOFF.Q THEN
       #Status := #STS_STOP;
   END_IF;
END_REGION

REGION Network 37: S120 EPOS - Force STATUS = STOP (Timeout SinaPos Mode not reached)
   RUNG wire#powerrail
      { S7_Templates := "SrcType := Int" } NE_Contact(in1 := #S120_SinaPos.ActMode, in2 := #MODE_5_SET_HOME_POSITION)
      { S7_Templates := "SrcType := Int" } EQ_Contact(in1 := #Status, in2 := #STS_DIRECT_HOME)
      wire#w1
      { S7_Templates := "time_type := Time" } #TON_ModeTimeOut.TON(pt := t#1500ms, et =>)
      Move(in := #STS_STOP, out1 => #Status)
   END_RUNG
   RUNG wire#powerrail
      { S7_Templates := "SrcType := Int" } NE_Contact(in1 := #S120_SinaPos.ActMode, in2 := #MODE_7_JOG)
      { S7_Templates := "SrcType := Int" } EQ_Contact(in1 := #Status, in2 := #STS_MOVE_VEL)
   END_RUNG wire#w1
   RUNG wire#powerrail
      { S7_Templates := "SrcType := Int" } NE_Contact(in1 := #S120_SinaPos.ActMode, in2 := #MODE_2_ABSOLUTE_POSITIONING)
      { S7_Templates := "SrcType := Int" } EQ_Contact(in1 := #Status, in2 := #STS_POSITIONING_START)
   END_RUNG wire#w1
   // the same network as SCL:
   #TON_ModeTimeOut(IN := ((#S120_SinaPos.ActMode <> #MODE_5_SET_HOME_POSITION) AND (#Status = #STS_DIRECT_HOME)) OR ((#S120_SinaPos.ActMode <> #MODE_7_JOG) AND (#Status = #STS_MOVE_VEL)) OR ((#S120_SinaPos.ActMode <> #MODE_2_ABSOLUTE_POSITIONING) AND (#Status = #STS_POSITIONING_START)),   // TON
                    PT := t#1500ms);
   IF #TON_ModeTimeOut.Q THEN #Status := #STS_STOP; END_IF;
END_REGION

REGION Network 38 (SCL): S120 EPOS - Control State Machine
   CASE #Status OF

           (* 
           //  ###############################################################################################
           //  STATUS = STOP
           // ###############################################################################################
           *)
       #STS_STOP:

           #S120_SinaPos.Jog1 := FALSE;
           #S120_SinaPos.Jog2 := FALSE;
           #S120_SinaPos.AxisRef := FALSE;
           #S120_SinaPos.ExecuteMode := FALSE;
           #S120_SinaPos.IntermediateStop := FALSE;


           IF NOT #S120_SinaPos.AxisEnabled AND NOT #S120_SinaPos.AxisError
           THEN
               #Status := #STS_0_IDLE;
           END_IF;

           (*    
           //  ###############################################################################################
           //  STATUS = IDLE
           // ###############################################################################################
           *)
       #STS_0_IDLE:


           #S120_SinaPos.Jog1 := FALSE;
           #S120_SinaPos.Jog2 := FALSE;
           #S120_SinaPos.AxisRef := FALSE;
           #S120_SinaPos.ExecuteMode := FALSE;
           #S120_SinaPos.IntermediateStop := FALSE;

           #WriteRefPos.Enable := FALSE;
           #Sts.S120.TargetApply := FALSE;


           IF #Ctrl.S120.Preset
           THEN
               #Status := #STS_DIRECT_HOME;

           ELSIF #Ctrl.S120.Jog_Minus OR #Ctrl.S120.Jog_Plus
           THEN
               #Status := #STS_MOVE_VEL;

           ELSIF #Ctrl.S120.Positioining OR #CIn.Manager.Control_ON
           THEN

               #Status := #STS_POSITIONING_START;

           END_IF;


           // Mode pos must have a valid value.Default is Mode 2
           // 
           IF #S120_SinaPos.ModePos < #MODE_1_RELATIVE_POSITIONING OR #S120_SinaPos.ModePos > #MODE_8_JOG_INCREMENTAL
           THEN
               #S120_SinaPos.ModePos := #MODE_2_ABSOLUTE_POSITIONING;
           END_IF;

           (*    
           //  ###############################################################################################
           //  STATUS = DIRECT HOME
           // ###############################################################################################
           *)

       #STS_DIRECT_HOME:

           #S120_SinaPos.ModePos := #MODE_5_SET_HOME_POSITION;
           //#S120_SinaPos.EnableAxis := TRUE;
           #WriteRefPos.Enable := TRUE;

           #S120_SinaPos.ExecuteMode := FALSE;

           IF (#S120_SinaPos.ActMode = #MODE_5_SET_HOME_POSITION)
               AND
               #WriteRefPos.Done
               AND 
               #Sts.Standstill
           THEN
               #WriteRefPos.Enable := FALSE;
               #S120_SinaPos.AxisRef := TRUE;
               #S120_SinaPos.ExecuteMode := TRUE;
           END_IF;


           (*    
           //  ###############################################################################################
           //  STATUS = MOVE VELOCITY
           // ###############################################################################################
           *)

       #STS_MOVE_VEL:

           #S120_SinaPos.ModePos := #MODE_7_JOG;
           #S120_SinaPos.EnableAxis := TRUE;
           #S120_SinaPos.CancelTraversing := TRUE;
           #S120_SinaPos.Jog1 := FALSE;
           #S120_SinaPos.Jog2 := FALSE;


           IF NOT #S120_SinaPos.AxisEnabled OR (#S120_SinaPos.ActMode <> #MODE_7_JOG)
           THEN
               ;
           ELSE
               #S120_SinaPos.Jog1 := #Ctrl.S120.Jog_Minus;
               #S120_SinaPos.Jog2 := #Ctrl.S120.Jog_Plus;
           END_IF;


           (*    
           //  ###############################################################################################
           //  STATUS = MOVE TO POSIITION
           // ###############################################################################################
           *)

       #STS_POSITIONING_START:

           #S120_SinaPos.ModePos := #MODE_2_ABSOLUTE_POSITIONING;
           #S120_SinaPos.EnableAxis := TRUE;
           #S120_SinaPos.CancelTraversing := TRUE;
           #S120_SinaPos.IntermediateStop := #Ctrl.S120.Positioining;


           // Convert target position from Eng.Unit To LU
           // 
           #Ctrl.S120.TargetPos := LREAL_TO_DINT(#Ctrl.Pos * 1000);


           IF (#Ctrl.S120.TargetPos <> #S120_SinaPos.Position)
               OR
               NOT #S120_SinaPos.AxisEnabled
               OR
               (#S120_SinaPos.ActMode <> #MODE_2_ABSOLUTE_POSITIONING)
           THEN
               #Sts.S120.TargetApply := FALSE;
           END_IF;


           #S120_SinaPos.ExecuteMode := FALSE;

           IF NOT #Sts.S120.TargetApply
               AND
               #S120_SinaPos.AxisEnabled
               AND
               (#S120_SinaPos.ActMode = #MODE_2_ABSOLUTE_POSITIONING)
           THEN

               #S120_SinaPos.ExecuteMode := TRUE;
               #S120_SinaPos.Position := #Ctrl.S120.TargetPos;
               #Sts.S120.TargetApply := TRUE;

           END_IF;


       ELSE
           #Status := #STS_STOP;

   END_CASE;
END_REGION

REGION Network 39: Reset enable Drive
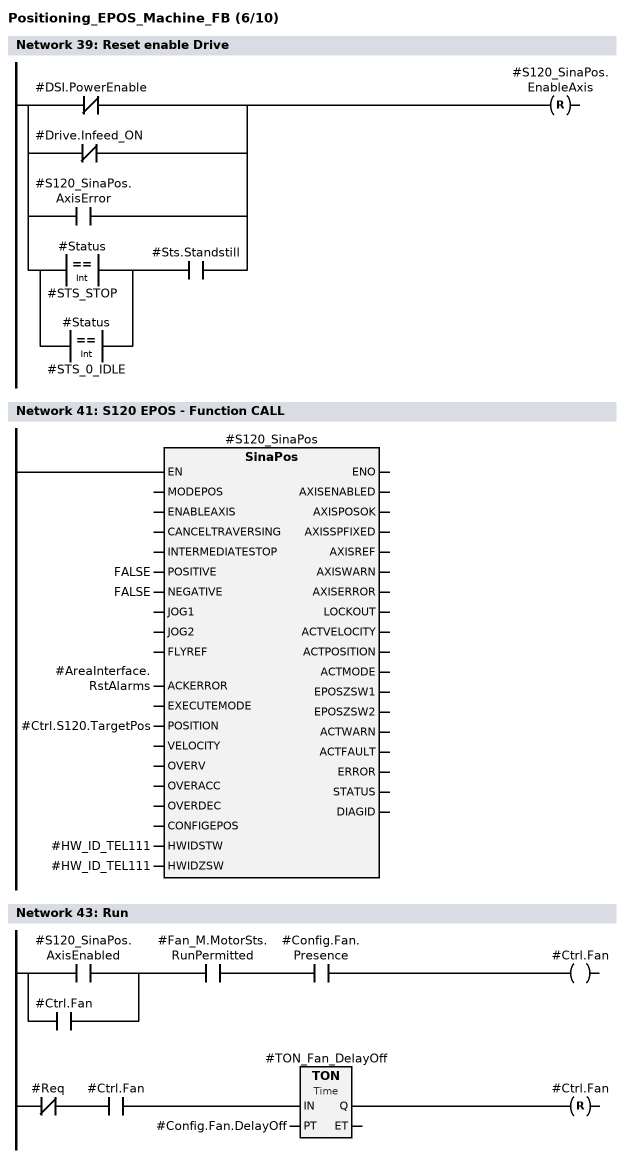
   RUNG wire#powerrail
      I_Contact( #DSI.PowerEnable )
      wire#w1
      R_Coil( #S120_SinaPos.EnableAxis )
   END_RUNG
   RUNG wire#powerrail
      I_Contact( #Drive.Infeed_ON )
   END_RUNG wire#w1
   RUNG wire#powerrail
      Contact( #S120_SinaPos.AxisError )
   END_RUNG wire#w1
   RUNG wire#powerrail
      { S7_Templates := "SrcType := Int" } EQ_Contact(in1 := #Status, in2 := #STS_STOP)
      wire#w2
      Contact( #Sts.Standstill )
   END_RUNG wire#w1
   RUNG wire#powerrail
      { S7_Templates := "SrcType := Int" } EQ_Contact(in1 := #Status, in2 := #STS_0_IDLE)
   END_RUNG wire#w2
   // the same network as SCL:
   IF NOT #DSI.PowerEnable OR NOT #Drive.Infeed_ON OR #S120_SinaPos.AxisError OR (((#Status = #STS_STOP) OR (#Status = #STS_0_IDLE)) AND #Sts.Standstill) THEN
       #S120_SinaPos.EnableAxis := FALSE;
   END_IF;
END_REGION

REGION Network 40 (SCL): S120 EPOS - Vel / Acc / Dec for MDI positioning
   // Coversione velocità in LU/min
   //
   #S120_SinaPos.Velocity := LREAL_TO_DINT(MIN_LREAL(IN1 := #Ctrl.Vel, IN2 := #Config.Ax.MaxVel_S120_P2571));
   #S120_SinaPos.Velocity := MAX_DINT(IN1 := #S120_SinaPos.Velocity, IN2 := 0);


   // Conversione acc/dec in %

   #S120_SinaPos.OverAcc := MIN_INT(IN1 := 100,IN2 :=  LREAL_TO_INT(#Ctrl.Acc / #Config.Ax.MaxAcc_S120_P2572 * 100.0));
   #S120_SinaPos.OverAcc := MAX_INT(IN1 := #S120_SinaPos.OverAcc, IN2 := 1);


   #S120_SinaPos.OverDec := MIN_INT(IN1 := 100, IN2 := LREAL_TO_INT(#Ctrl.Dec / #Config.Ax.MaxDec_S120_P2573 * 100.0));
   #S120_SinaPos.OverDec := MAX_INT(IN1 := #S120_SinaPos.OverDec, IN2 := 1);


   // Velocity override
   // 

   #S120_SinaPos.OverV := 100;

   IF #CIn.VelocityOverride.Enable THEN
       #S120_SinaPos.OverV := LREAL_TO_INT(#CIn.VelocityOverride.Value);
   END_IF;


   //Reference position

   #WriteRefPos(ReadWrite := 1,
                 ParNo := 2599,
                 Index := 0,
                 AxisNo := #Drive.AxisID,
                 HW_ID := #Drive.AccessPoint,
                 TokenChain := #Drive.TokenChain,
                 ValueWriteDint := LREAL_TO_DINT(#HMI.PresetPosition * 1000.0));
END_REGION

REGION Network 41: S120 EPOS - Function CALL
   RUNG wire#powerrail
      #S120_SinaPos.SinaPos(ModePos :=, EnableAxis :=, CancelTraversing :=, IntermediateStop :=, Positive := FALSE, Negative := FALSE, Jog1 :=, Jog2 :=, FlyRef :=, AckError := #AreaInterface.RstAlarms, ExecuteMode :=, Position := #Ctrl.S120.TargetPos, Velocity :=, OverV :=, OverAcc :=, OverDec :=, ConfigEPos :=, HWIDSTW := #HW_ID_TEL111, HWIDZSW := #HW_ID_TEL111, AxisEnabled =>, AxisPosOk =>, AxisSpFixed =>, AxisRef =>, AxisWarn =>, AxisError =>, Lockout =>, ActVelocity =>, ActPosition =>, ActMode =>, EPosZSW1 =>, EPosZSW2 =>, ActWarn =>, ActFault =>, Error =>, Status =>, DiagId =>)
   END_RUNG
   // the same network as SCL:
   #S120_SinaPos(Positive := FALSE,   // SinaPos
                 Negative := FALSE,
                 AckError := #AreaInterface.RstAlarms,
                 Position := #Ctrl.S120.TargetPos,
                 HWIDSTW := #HW_ID_TEL111,
                 HWIDZSW := #HW_ID_TEL111);
END_REGION

REGION Network 42: <<< MOTOR FAN >>>
END_REGION

REGION Network 43: Run
   RUNG wire#powerrail
      Contact( #S120_SinaPos.AxisEnabled )
      wire#w1
      Contact( #Fan_M.MotorSts.RunPermitted )
      Contact( #Config.Fan.Presence )
      Coil( #Ctrl.Fan )
   END_RUNG
   RUNG wire#powerrail
      Contact( #Ctrl.Fan )
   END_RUNG wire#w1
   RUNG wire#powerrail
      I_Contact( #Req )
      Contact( #Ctrl.Fan )
      { S7_Templates := "time_type := Time" } #TON_Fan_DelayOff.TON(pt := #Config.Fan.DelayOff, et =>)
      R_Coil( #Ctrl.Fan )
   END_RUNG
   // the same network as SCL:
   #Ctrl.Fan := (#S120_SinaPos.AxisEnabled OR #Ctrl.Fan) AND #Fan_M.MotorSts.RunPermitted AND #Config.Fan.Presence;
   #TON_Fan_DelayOff(IN := NOT #Req AND #Ctrl.Fan, PT := #Config.Fan.DelayOff);   // TON
   IF #TON_Fan_DelayOff.Q THEN #Ctrl.Fan := FALSE; END_IF;
END_REGION

REGION Network 44: Device
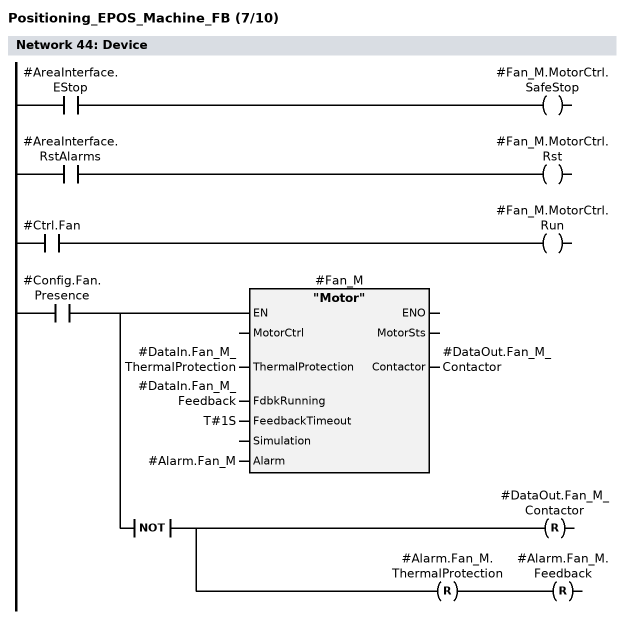
   RUNG wire#powerrail
      Contact( #AreaInterface.EStop )
      Coil( #Fan_M.MotorCtrl.SafeStop )
   END_RUNG
   RUNG wire#powerrail
      Contact( #AreaInterface.RstAlarms )
      Coil( #Fan_M.MotorCtrl.Rst )
   END_RUNG
   RUNG wire#powerrail
      Contact( #Ctrl.Fan )
      Coil( #Fan_M.MotorCtrl.Run )
   END_RUNG
   RUNG wire#powerrail
      Contact( #Config.Fan.Presence )
      wire#w1
      #Fan_M(MotorCtrl :=, ThermalProtection := #DataIn.Fan_M_ThermalProtection, FdbkRunning := #DataIn.Fan_M_Feedback, FeedbackTimeout := T#1S, Simulation :=, Alarm := #Alarm.Fan_M, MotorSts =>, Contactor => #DataOut.Fan_M_Contactor)
   END_RUNG
   RUNG wire#w1
      Not()
      wire#w2
      R_Coil( #DataOut.Fan_M_Contactor )
   END_RUNG
   RUNG wire#w2
      R_Coil( #Alarm.Fan_M.ThermalProtection )
      R_Coil( #Alarm.Fan_M.Feedback )
   END_RUNG
   // the same network as SCL:
   #Fan_M.MotorCtrl.SafeStop := #AreaInterface.EStop;
   #Fan_M.MotorCtrl.Rst := #AreaInterface.RstAlarms;
   #Fan_M.MotorCtrl.Run := #Ctrl.Fan;
   IF #Config.Fan.Presence THEN
       #Fan_M(ThermalProtection := #DataIn.Fan_M_ThermalProtection,   // "Motor"
              FdbkRunning := #DataIn.Fan_M_Feedback,
              FeedbackTimeout := T#1S,
              Alarm := #Alarm.Fan_M,
              Contactor => #DataOut.Fan_M_Contactor);
   END_IF;
   IF NOT #Config.Fan.Presence THEN
       #DataOut.Fan_M_Contactor := FALSE;
       #Alarm.Fan_M.ThermalProtection := FALSE;
       #Alarm.Fan_M.Feedback := FALSE;
   END_IF;
END_REGION

REGION Network 45: >
END_REGION

REGION Network 46: >
END_REGION

REGION Network 47: Coordination Out
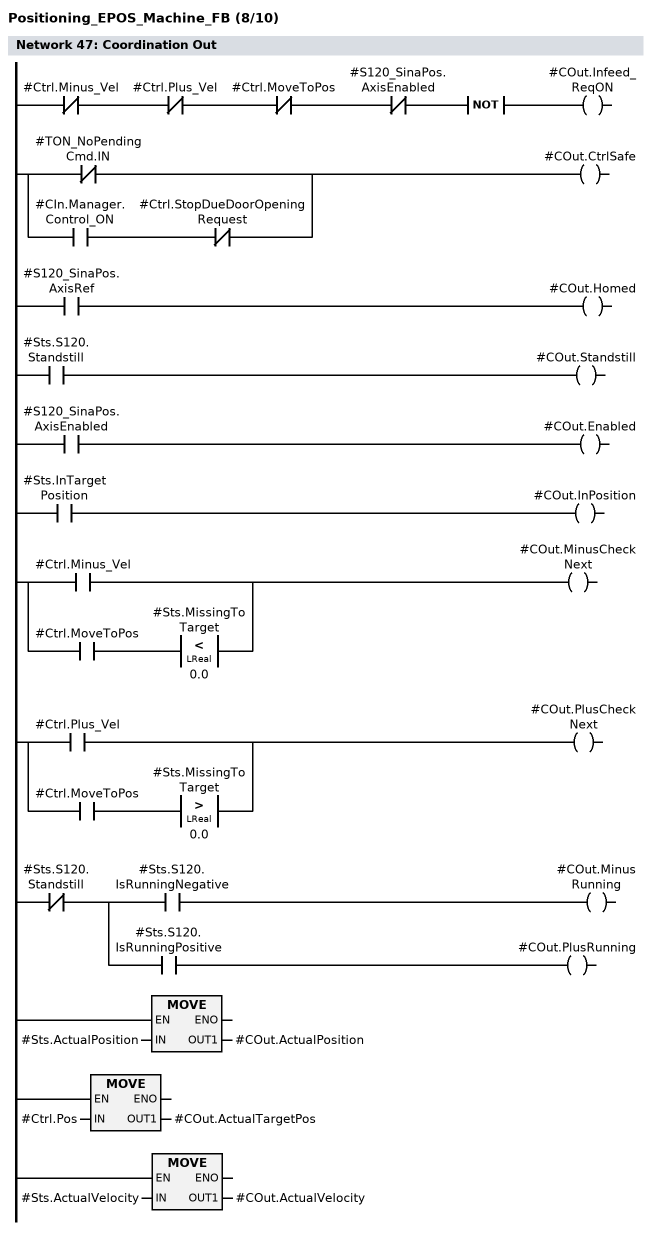
   RUNG wire#powerrail
      I_Contact( #Ctrl.Minus_Vel )
      I_Contact( #Ctrl.Plus_Vel )
      I_Contact( #Ctrl.MoveToPos )
      I_Contact( #S120_SinaPos.AxisEnabled )
      Not()
      Coil( #COut.Infeed_ReqON )
   END_RUNG
   RUNG wire#powerrail
      I_Contact( #TON_NoPendingCmd.IN )
      wire#w1
      Coil( #COut.CtrlSafe )
   END_RUNG
   RUNG wire#powerrail
      Contact( #CIn.Manager.Control_ON )
      I_Contact( #Ctrl.StopDueDoorOpeningRequest )
   END_RUNG wire#w1
   RUNG wire#powerrail
      Contact( #S120_SinaPos.AxisRef )
      Coil( #COut.Homed )
   END_RUNG
   RUNG wire#powerrail
      Contact( #Sts.S120.Standstill )
      Coil( #COut.Standstill )
   END_RUNG
   RUNG wire#powerrail
      Contact( #S120_SinaPos.AxisEnabled )
      Coil( #COut.Enabled )
   END_RUNG
   RUNG wire#powerrail
      Contact( #Sts.InTargetPosition )
      Coil( #COut.InPosition )
   END_RUNG
   RUNG wire#powerrail
      Contact( #Ctrl.Minus_Vel )
      wire#w2
      Coil( #COut.MinusCheckNext )
   END_RUNG
   RUNG wire#powerrail
      Contact( #Ctrl.MoveToPos )
      { S7_Templates := "SrcType := LReal" } LT_Contact(in1 := #Sts.MissingToTarget, in2 := 0.0)
   END_RUNG wire#w2
   RUNG wire#powerrail
      Contact( #Ctrl.Plus_Vel )
      wire#w3
      Coil( #COut.PlusCheckNext )
   END_RUNG
   RUNG wire#powerrail
      Contact( #Ctrl.MoveToPos )
      { S7_Templates := "SrcType := LReal" } GT_Contact(in1 := #Sts.MissingToTarget, in2 := 0.0)
   END_RUNG wire#w3
   RUNG wire#powerrail
      I_Contact( #Sts.S120.Standstill )
      wire#w4
      Contact( #Sts.S120.IsRunningNegative )
      Coil( #COut.MinusRunning )
   END_RUNG
   RUNG wire#w4
      Contact( #Sts.S120.IsRunningPositive )
      Coil( #COut.PlusRunning )
   END_RUNG
   RUNG wire#powerrail
      Move(in := #Sts.ActualPosition, out1 => #COut.ActualPosition)
   END_RUNG
   RUNG wire#powerrail
      Move(in := #Ctrl.Pos, out1 => #COut.ActualTargetPos)
   END_RUNG
   RUNG wire#powerrail
      Move(in := #Sts.ActualVelocity, out1 => #COut.ActualVelocity)
   END_RUNG
   // the same network as SCL:
   #COut.Infeed_ReqON := NOT (NOT #Ctrl.Minus_Vel AND NOT #Ctrl.Plus_Vel AND NOT #Ctrl.MoveToPos AND NOT #S120_SinaPos.AxisEnabled);
   #COut.CtrlSafe := NOT #TON_NoPendingCmd.IN OR (#CIn.Manager.Control_ON AND NOT #Ctrl.StopDueDoorOpeningRequest);
   #COut.Homed := #S120_SinaPos.AxisRef;
   #COut.Standstill := #Sts.S120.Standstill;
   #COut.Enabled := #S120_SinaPos.AxisEnabled;
   #COut.InPosition := #Sts.InTargetPosition;
   #COut.MinusCheckNext := #Ctrl.Minus_Vel OR (#Ctrl.MoveToPos AND (#Sts.MissingToTarget < 0.0));
   #COut.PlusCheckNext := #Ctrl.Plus_Vel OR (#Ctrl.MoveToPos AND (#Sts.MissingToTarget > 0.0));
   #COut.MinusRunning := NOT #Sts.S120.Standstill AND #Sts.S120.IsRunningNegative;
   #COut.PlusRunning := NOT #Sts.S120.Standstill AND #Sts.S120.IsRunningPositive;
   #COut.ActualPosition := #Sts.ActualPosition;
   #COut.ActualTargetPos := #Ctrl.Pos;
   #COut.ActualVelocity := #Sts.ActualVelocity;
END_REGION

REGION Network 48: Warning Missing conditions
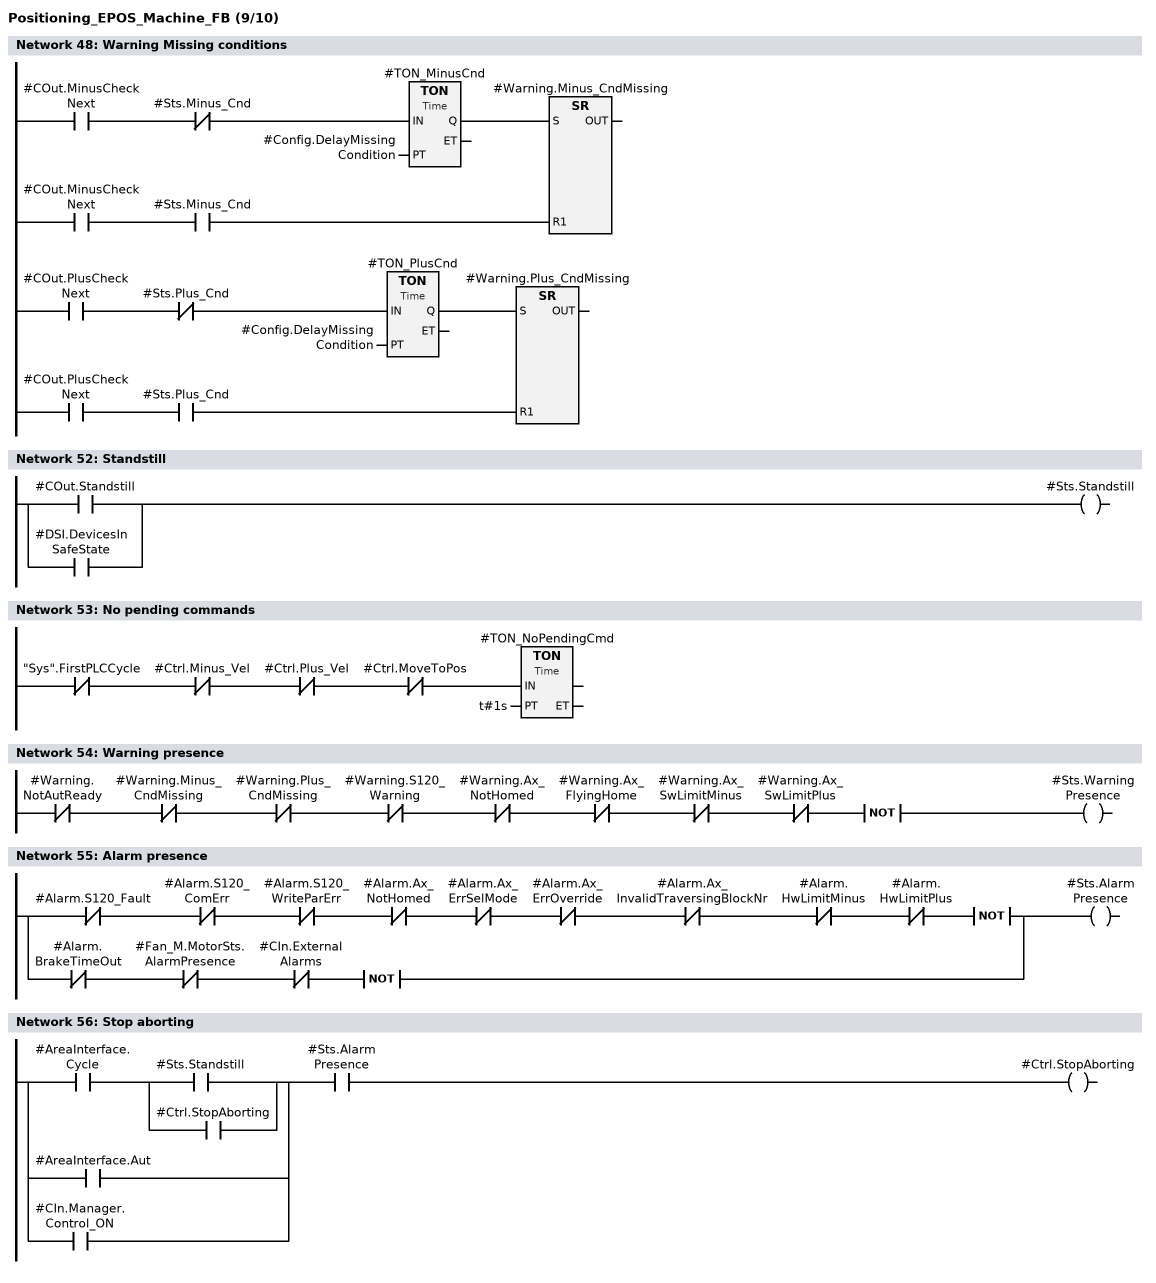
   RUNG wire#powerrail
      Contact( #COut.MinusCheckNext )
      I_Contact( #Sts.Minus_Cnd )
      { S7_Templates := "time_type := Time" } #TON_MinusCnd.TON(pt := #Config.DelayMissingCondition, et =>)
      S_SR(operand := #Warning.Minus_CndMissing, r1 := wire#w1)
   END_RUNG
   RUNG wire#powerrail
      Contact( #COut.MinusCheckNext )
      Contact( #Sts.Minus_Cnd )
   END_RUNG wire#w1
   RUNG wire#powerrail
      Contact( #COut.PlusCheckNext )
      I_Contact( #Sts.Plus_Cnd )
      { S7_Templates := "time_type := Time" } #TON_PlusCnd.TON(pt := #Config.DelayMissingCondition, et =>)
      S_SR(operand := #Warning.Plus_CndMissing, r1 := wire#w2)
   END_RUNG
   RUNG wire#powerrail
      Contact( #COut.PlusCheckNext )
      Contact( #Sts.Plus_Cnd )
   END_RUNG wire#w2
   // the same network as SCL:
   #TON_MinusCnd(IN := #COut.MinusCheckNext AND NOT #Sts.Minus_Cnd, PT := #Config.DelayMissingCondition);   // TON
   IF #TON_MinusCnd.Q THEN
       #Warning.Minus_CndMissing := TRUE;   // SR flip-flop
   END_IF;
   IF #COut.MinusCheckNext AND #Sts.Minus_Cnd THEN #Warning.Minus_CndMissing := FALSE; END_IF;
   #TON_PlusCnd(IN := #COut.PlusCheckNext AND NOT #Sts.Plus_Cnd, PT := #Config.DelayMissingCondition);   // TON
   IF #TON_PlusCnd.Q THEN
       #Warning.Plus_CndMissing := TRUE;   // SR flip-flop
   END_IF;
   IF #COut.PlusCheckNext AND #Sts.Plus_Cnd THEN #Warning.Plus_CndMissing := FALSE; END_IF;
END_REGION

REGION Network 49: >
END_REGION

REGION Network 50: >
END_REGION

REGION Network 51: <<< MACHINE STATUS >>>
END_REGION

REGION Network 52: Standstill
   RUNG wire#powerrail
      Contact( #COut.Standstill )
      wire#w1
      Coil( #Sts.Standstill )
   END_RUNG
   RUNG wire#powerrail
      Contact( #DSI.DevicesInSafeState )
   END_RUNG wire#w1
   // the same network as SCL:
   #Sts.Standstill := #COut.Standstill OR #DSI.DevicesInSafeState;
END_REGION

REGION Network 53: No pending commands
   RUNG wire#powerrail
      I_Contact( "Sys".FirstPLCCycle )
      I_Contact( #Ctrl.Minus_Vel )
      I_Contact( #Ctrl.Plus_Vel )
      I_Contact( #Ctrl.MoveToPos )
      { S7_Templates := "time_type := Time" } #TON_NoPendingCmd.TON(pt := t#1s, et =>)
   END_RUNG
   // the same network as SCL:
   #TON_NoPendingCmd(IN := NOT "Sys".FirstPLCCycle AND NOT #Ctrl.Minus_Vel AND NOT #Ctrl.Plus_Vel AND NOT #Ctrl.MoveToPos,   // TON
                     PT := t#1s);
END_REGION

REGION Network 54: Warning presence
   RUNG wire#powerrail
      I_Contact( #Warning.NotAutReady )
      I_Contact( #Warning.Minus_CndMissing )
      I_Contact( #Warning.Plus_CndMissing )
      I_Contact( #Warning.S120_Warning )
      I_Contact( #Warning.Ax_NotHomed )
      I_Contact( #Warning.Ax_FlyingHome )
      I_Contact( #Warning.Ax_SwLimitMinus )
      I_Contact( #Warning.Ax_SwLimitPlus )
      Not()
      Coil( #Sts.WarningPresence )
   END_RUNG
   // the same network as SCL:
   #Sts.WarningPresence := NOT (NOT #Warning.NotAutReady AND NOT #Warning.Minus_CndMissing AND NOT #Warning.Plus_CndMissing AND NOT #Warning.S120_Warning AND NOT #Warning.Ax_NotHomed AND NOT #Warning.Ax_FlyingHome AND NOT #Warning.Ax_SwLimitMinus AND NOT #Warning.Ax_SwLimitPlus);
END_REGION

REGION Network 55: Alarm presence
   RUNG wire#powerrail
      I_Contact( #Alarm.S120_Fault )
      I_Contact( #Alarm.S120_ComErr )
      I_Contact( #Alarm.S120_WriteParErr )
      I_Contact( #Alarm.Ax_NotHomed )
      I_Contact( #Alarm.Ax_ErrSelMode )
      I_Contact( #Alarm.Ax_ErrOverride )
      I_Contact( #Alarm.Ax_InvalidTraversingBlockNr )
      I_Contact( #Alarm.HwLimitMinus )
      I_Contact( #Alarm.HwLimitPlus )
      Not()
      wire#w1
      Coil( #Sts.AlarmPresence )
   END_RUNG
   RUNG wire#powerrail
      I_Contact( #Alarm.BrakeTimeOut )
      I_Contact( #Fan_M.MotorSts.AlarmPresence )
      I_Contact( #CIn.ExternalAlarms )
      Not()
   END_RUNG wire#w1
   // the same network as SCL:
   #Sts.AlarmPresence := NOT (NOT #Alarm.S120_Fault AND NOT #Alarm.S120_ComErr AND NOT #Alarm.S120_WriteParErr AND NOT #Alarm.Ax_NotHomed AND NOT #Alarm.Ax_ErrSelMode AND NOT #Alarm.Ax_ErrOverride AND NOT #Alarm.Ax_InvalidTraversingBlockNr AND NOT #Alarm.HwLimitMinus AND NOT #Alarm.HwLimitPlus) OR NOT (NOT #Alarm.BrakeTimeOut AND NOT #Fan_M.MotorSts.AlarmPresence AND NOT #CIn.ExternalAlarms);
END_REGION

REGION Network 56: Stop aborting
   RUNG wire#powerrail
      Contact( #AreaInterface.Cycle )
      wire#w1
      Contact( #Sts.Standstill )
      wire#w2
      Contact( #Sts.AlarmPresence )
      Coil( #Ctrl.StopAborting )
   END_RUNG
   RUNG wire#w1
      Contact( #Ctrl.StopAborting )
   END_RUNG wire#w2
   RUNG wire#powerrail
      Contact( #AreaInterface.Aut )
   END_RUNG wire#w2
   RUNG wire#powerrail
      Contact( #CIn.Manager.Control_ON )
   END_RUNG wire#w2
   // the same network as SCL:
   #Ctrl.StopAborting := ((#AreaInterface.Cycle AND (#Sts.Standstill OR #Ctrl.StopAborting)) OR #AreaInterface.Aut OR #CIn.Manager.Control_ON) AND #Sts.AlarmPresence;
END_REGION

REGION Network 57 (SCL): Collect machine to zone interface
   #MachineInterface.AutReady := #AreaInterface.Aut AND NOT #Sts.AlarmPresence;
   #MachineInterface.Aborting := #Ctrl.StopAborting;
   #MachineInterface.MotionsStandStill := #TON_NoPendingCmd.Q AND #Sts.Standstill;
   #MachineInterface.AckStopInPhase := #Ctrl.StopInPhase AND #MachineInterface.MotionsStandStill;
   #MachineInterface.AckStopProgrammed := #Ctrl.StopProgrammed AND #MachineInterface.MotionsStandStill;
   #MachineInterface.AlarmsPresence := #Sts.AlarmPresence;
   #MachineInterface.WarningPresence := #Sts.WarningPresence;
END_REGION

REGION Network 58: Warning Machine not ready for automatic
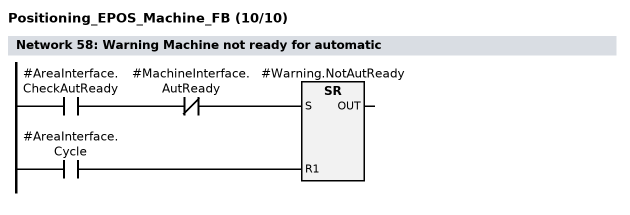
   RUNG wire#powerrail
      Contact( #AreaInterface.CheckAutReady )
      I_Contact( #MachineInterface.AutReady )
      S_SR(operand := #Warning.NotAutReady, r1 := wire#w1)
   END_RUNG
   RUNG wire#powerrail
      Contact( #AreaInterface.Cycle )
   END_RUNG wire#w1
   // the same network as SCL:
   IF #AreaInterface.CheckAutReady AND NOT #MachineInterface.AutReady THEN
       #Warning.NotAutReady := TRUE;   // SR flip-flop
   END_IF;
   IF #AreaInterface.Cycle THEN #Warning.NotAutReady := FALSE; END_IF;
END_REGION

REGION Network 59: +
END_REGION

REGION Network 60 (SCL): HMI Status Positioning EPOS Machine
   // Area dati Status per HMI sull'azionamento

   #HMI.Sts.Enabled := #S120_SinaPos.AxisEnabled;
   #HMI.Sts.Standstill := #Sts.Standstill;
   #HMI.Sts.Homed := #COut.Homed;
   #HMI.Sts.Alarm := #Sts.AlarmPresence;
   #HMI.Sts.Warning := #Sts.WarningPresence;
   #HMI.Sts.Plus_Run := #COut.PlusRunning;
   #HMI.Sts.Minus_Run := #COut.MinusRunning;
   #HMI.Sts.InTargetPos := #Sts.InTargetPosition;
   #HMI.Sts.MinPosReached := #COut.MinusLsSwReached OR #COut.MinusLimitReached;
   #HMI.Sts.MaxPosReached := #COut.PlusLsSwReached OR #COut.PlusLimitReached;
   #HMI.Sts.TargetPos := #COut.ActualTargetPos;
   #HMI.Sts.ActualPos := #COut.ActualPosition;
   #HMI.Sts.ActualVel := #COut.ActualVelocity;
END_REGION

REGION Network 61: +
END_REGION

REGION Network 62: +
END_REGION
END_FUNCTION_BLOCK
